// TwinCAT 3 PLC project PLC
// ProgramVersion: 3.1.4022.1
// libraries:
//   Tc2_Standard, * (Beckhoff Automation GmbH)
//   Tc2_System, * (Beckhoff Automation GmbH)
//   Tc3_Module, * (Beckhoff Automation GmbH)
// project tree:
//   DUTs/ Trapez.TcDUT, Trig.TcDUT
//   / GlobalTextList.TcGTLO, PlcTask.TcTTO, Visualization Manager.TcVMO (not stored)
//   GVLs/ IO.TcGVL, Temperatures.TcGVL
//   POUs/Fuzzy/ fbFuzzyController.TcPOU, FuzzificationTrapez.TcPOU, FuzzificationTrig.TcPOU
//   POUs/ MAIN.TcPOU, SLL.TcPOU
//   POUs/PID/ fbFlowControl.TcPOU, fbPIContoller.TcPOU, fbTempControl.TcPOU
//   POUs/utils/ fbB2U.TcPOU, fbIfElse.TcPOU, fbScale.TcPOU, fbSplit.TcPOU, fbU2B.TcPOU
// real-time tasks:
//   TASK PlcTask: cycle T#10ms, priority 20, ADS port 350
// I/O:
//   DEVICE Device 3 (EtherCAT), AmsNetId 192.168.8.100.4.1
//     Box 1 (ABB CI511) [CI511-ETHCAT (4AI 2AO 8DI 8DO)]
//     Box 2 (ABB CI512) [CI512-ETHCAT (8DC 8DI 8DO)]
// variable links:
//   PLC/PLC Instance <-> Device 3 (EtherCAT)/Box 1 (ABB CI511)
//     PlcTask Inputs/IO.AI0_Temp <-> Inputs/AI 0
//     PlcTask Inputs/IO.AI1_Pres <-> Inputs/AI 1
//     PlcTask Outputs/IO.AO0_Fan <-> Outputs/AO 0
//     PlcTask Outputs/IO.AO1_Heater <-> Outputs/AO 1
//   PLC/PLC Instance <-> Device 3 (EtherCAT)/Box 2 (ABB CI512)
//     PlcTask Inputs/IO.DI_SLL <-> Inputs/DI
//     PlcTask Outputs/IO.DO_SLL <-> Outputs/DO

CONFIGURATION PLC
    RESOURCE PLC ON TwinCAT3
        TASK PlcTask(INTERVAL := T#10ms, PRIORITY := 20);
        PROGRAM MAIN WITH PlcTask : MAIN;
    END_RESOURCE
END_CONFIGURATION

// ---- DUTs/Trapez.TcDUT
TYPE Trapez :
STRUCT
	A	:REAL;
	B	:REAL;
	C	:REAL;
	D	:REAL;
END_STRUCT
END_TYPE

// ---- DUTs/Trig.TcDUT
TYPE Trig :
STRUCT
	A	:REAL;
	B	:REAL;
	C	:REAL;
END_STRUCT
END_TYPE

// ---- GVLs/IO.TcGVL
{attribute 'qualified_only'}
VAR_GLOBAL
	AI0_Temp 	AT %I*: INT;	//Temperature
	AI1_Pres 	AT %I*:	INT;	//Pressure
	AO0_Fan 	AT %Q*: INT;	//Fan
	AO1_Heater	AT %Q*:	INT;	//Heater
	DI_SLL		AT %I*: UINT;	//Digital input
	DO_SLL		AT %Q*: UINT;	//Digital output	
END_VAR

// ---- GVLs/Temperatures.TcGVL
{attribute 'qualified_only'}
VAR_GLOBAL
	T_Ref	:REAL := 40;
	T_Act	:REAL;
END_VAR

// ---- POUs/MAIN.TcPOU
PROGRAM MAIN
VAR
	HeaterRatio			:REAL	:= 20;
	FanRatio			:REAL;
	Region				:REAL	:= 2.5; //Allowed error +- for the steady-state
	
	fbTempScale			:fbScale;
	fbFControl			:fbFuzzyController;
	fbPIControl			:fbPIContoller;
	
	Timer				:TON;
END_VAR

//Handle digital I/O
SLL(SteadyStateRegion := Region);

//HeaterRatio can be cnaged from the GUI
IO.AO1_Heater := REAL_TO_INT(27468 * HeaterRatio/100);
//Used in the GUI
FanRatio := INT_TO_REAL(IO.AO0_Fan)/INT_TO_REAL(27468)*100;


//Run the controller
//Controller can be switched between PI and Fuzzy
IF SLL.ControllerSwitch THEN
	//Longer samplingtime allows error to accumulate
	//10ms had too small changes between samples
	Timer(IN := NOT Timer.Q, PT := T#0.1S);
	IF Timer.Q THEN
		fbFControl(On := SLL.ControllerOn);
	END_IF
ELSE
	fbPIControl(On := SLL.ControllerOn);
END_IF

//Current temperature as celsius
fbTempScale(IN := IO.AI0_Temp, Scale_L := 20, Scale_H := 120);
Temperatures.T_Act := fbTempScale.OUT;

END_PROGRAM

// ---- POUs/utils/fbScale.TcPOU
FUNCTION_BLOCK fbScale
VAR_INPUT
	IN		:REAL;
	Scale_L	:REAL;
	Scale_H	:REAL;
	bType	:BOOL	:=TRUE;	//TRUE = analog val to real, FALSE = real to analog
END_VAR
VAR_OUTPUT
	OUT		:REAL;
END_VAR
VAR
	AnalogMax :REAL := 27648;
END_VAR

IF bType THEN
	OUT := IN / AnalogMax * (Scale_H - Scale_L) + Scale_L;
ELSE
	OUT := (AnalogMax * (IN - Scale_L)) / (Scale_H - Scale_L);
END_IF

END_FUNCTION_BLOCK

// ---- POUs/Fuzzy/fbFuzzyController.TcPOU
FUNCTION_BLOCK fbFuzzyController
VAR_INPUT
	On					:BOOL;
END_VAR
VAR_OUTPUT
END_VAR
VAR
	HOT, COLD						:Trapez;
	WARM, COOL						:Trig;
	
	DECREASING, INCREASING			:Trapez;
	SLOWDOWN, SPEEDUP				:Trig;
	
	Temperature						:REAL;
	Temp_prev						:REAL := 0;
	Error							:REAL := 0;
	
	//Degree of membership
	Hot_h, Warm_h, Cool_h, Cold_h	:REAL;
	Decreasing_h, Increasing_h		:REAL;
	
	Rule, Rule1, Rule2, Rule3, Rule4, Rule5, Rule6 :REAL;
	
	u	:REAL;
	Fan_R	:REAL;
	Scale	:REAL := 0.1;
END_VAR

//If controller is switched off, turn the fan off and reset the controllers
IF NOT On THEN
	IO.AO0_Fan := 0;
	RETURN;
END_IF

//Temperature
HOT.A := -100; HOT.B := -100; HOT.C := -5; HOT.D := -0.5;
WARM.A := -5; WARM.B := -2.5; WARM.C := 0;
COOL.A := 0; COOL.B := 2.5; COOL.C := 5;
COLD.A := 0.5; COLD.B := 5; COLD.C := 100; COLD.D := 100;

//Error
DECREASING.A := -0.1; DECREASING.B := -0.03; DECREASING.C := -0.0006; DECREASING.D := 0;
INCREASING.A := 0; INCREASING.B := 0.0006; INCREASING.C := 0.03; INCREASING.D := 0.1;

//Control signal
SLOWDOWN.A := 1; SLOWDOWN.B := -1; SLOWDOWN.C := -1;
SPEEDUP.A := -1; SPEEDUP.B := 1; SPEEDUP.C := 1;

//Controller inputs
Temperature := Temperatures.T_Ref - Temperatures.T_Act;
Error := Temp_prev - Temperature;
Temp_prev := Temperature;

//Fuzzification
Hot_h := FuzzificationTrapez(Temperature, HOT);
Cold_h := FuzzificationTrapez(Temperature, COLD);
Warm_h := FuzzificationTrig(Temperature, WARM);
Cool_h := FuzzificationTrig(Temperature, Cool);
Decreasing_h := FuzzificationTrapez(Error, DECREASING);
Increasing_h := FuzzificationTrapez(Error, INCREASING);

//Rules
//IF Temperature IS Hot
IF Hot_h > 0 THEN
	Rule1 := Hot_h;
END_IF
//IF Temperature IS Warm AND Error IS Increasing
IF Warm_h > 0 AND Increasing_h > 0 THEN
	Rule2 := MIN(Warm_h,Increasing_h);
END_IF
//IF Temperature IS Warm AND Error IS Decreasing
IF Warm_h > 0 AND Decreasing_h > 0 THEN
	Rule3 := MIN(Warm_h,Decreasing_h);
END_IF
//IF Temperature IS Cool AND Error IS Increasing
IF Cool_h > 0 AND Increasing_h > 0 THEN
	Rule4 := MIN(Cool_h,Increasing_h);
END_IF
//IF Temperature IS Cool AND Error IS Decreasing
IF Cool_h > 0 AND Decreasing_h > 0 THEN
	Rule5 := MIN(Cool_h,Decreasing_h);
END_IF
//IF Temperature IS Cold
IF Cold_h > 0 THEN
	Rule6 := Cold_h;
END_IF

//Rule with the max value is the most significant
Rule := MAX(Rule1,Rule2,Rule3,Rule4,Rule5,Rule6);

//Defuzzification using Mean of Max.
//Boundaries with alpha-cut at max rule's degree
IF Rule = Rule1 OR Rule = Rule2 OR Rule = Rule4 THEN
	u := ((SPEEDUP.B-SPEEDUP.A)*Rule+SPEEDUP.A + (-(SPEEDUP.C-SPEEDUP.B)*Rule+SPEEDUP.C))/2;
ELSIF Rule = Rule3 OR Rule = Rule5 OR Rule = Rule6 THEN
	u := ((SLOWDOWN.B-SLOWDOWN.A)*Rule+SLOWDOWN.A + (-(SLOWDOWN.C-SLOWDOWN.B)*Rule+SLOWDOWN.C))/2;
END_IF
//Resetting values to zero for the next execution
Rule1 := Rule2 := Rule3 := Rule4 := Rule5 := Rule6 := 0;

//Calculating the new fan usage 0-100
Fan_R := Fan_R + u * Scale;
IF Fan_R > 100 THEN
	Fan_R := 100;
ELSIF FAN_R < 0 THEN
	Fan_R := 0;
END_IF

IO.AO0_Fan := REAL_TO_INT(27648*Fan_R/100);

END_FUNCTION_BLOCK

// ---- POUs/Fuzzy/FuzzificationTrapez.TcPOU
FUNCTION FuzzificationTrapez : REAL
VAR_INPUT
	x		:REAL;
	trapez	:Trapez;
END_VAR
VAR
END_VAR

IF x <= trapez.A THEN
	FuzzificationTrapez := 0;
ELSIF trapez.A < x AND x <= trapez.B THEN
	FuzzificationTrapez := (x-trapez.A)/(trapez.B-trapez.A);
ELSIF trapez.B <= x AND x <= trapez.C THEN
	FuzzificationTrapez := 1;
ELSIF trapez.C < x AND x <= trapez.D THEN
	FuzzificationTrapez := (trapez.D-x)/(trapez.D-trapez.C);
ELSIF trapez.D < x THEN
	FuzzificationTrapez := 0; 
END_IF

END_FUNCTION

// ---- POUs/Fuzzy/FuzzificationTrig.TcPOU
FUNCTION FuzzificationTrig : REAL
VAR_INPUT
	x		:REAL;
	trig	:Trig;
END_VAR
VAR
END_VAR

IF x <= trig.A THEN
	FuzzificationTrig := 0;
ELSIF trig.A < x AND x <= trig.B THEN
	FuzzificationTrig := (x-trig.A)/(trig.B-trig.A);
ELSIF trig.B < x AND x <= trig.C THEN
	FuzzificationTrig := (trig.C-x)/(trig.C-trig.B);
ELSIF trig.C < x THEN
	FuzzificationTrig := 0; 
END_IF

END_FUNCTION

// ---- POUs/PID/fbPIContoller.TcPOU
FUNCTION_BLOCK fbPIContoller
VAR_INPUT
	On					:BOOL;
END_VAR
VAR
	//PID-variables
	P_Temperature		:REAL	:= 10.0;
	P_Flow				:REAL	:= 2.0;
	Ki_Temperature		:REAL 	:= 0.005;
	Ki_Flow				:REAL 	:= 0.001;
	I_CapTemperature	:INT	:= 80;
	I_CapFlow			:INT	:= 80;

	//FBs

	fbFlowScale			:fbScale;
	fbFlowP2AScale		:fbScale;
	
	fbFlowController	:fbFlowControl;
	fbTempController	:fbTempControl;
END_VAR

//If controller is switched off, turn the fan off and reset the controllers
IF NOT On THEN
	IO.AO0_Fan := 0;
	RETURN;
END_IF

//Current flowrate
fbFlowScale(IN := IO.AI1_Pres, Scale_L := 0, Scale_H := 100);

fbTempController(
	Act := Temperatures.T_Act,
	Ref := Temperatures.T_Ref,
	Kp := P_Temperature,
	Ki := Ki_Temperature,
	I_Cap := I_CapTemperature);

fbFlowController(
	Act := fbFlowScale.OUT,
	Ref := fbTempController.OUT,
	Kp := P_Flow,
	Ki := Ki_Flow,
	I_Cap := I_CapFlow);

//Percentage to analog value (0-100% -> 0-27468)
fbFlowP2AScale(IN := fbFlowController.OUT, Scale_L := 0, Scale_H := 100, bType := FALSE);
IO.AO0_Fan := REAL_TO_INT(fbFlowP2AScale.OUT);

END_FUNCTION_BLOCK

// ---- POUs/PID/fbFlowControl.TcPOU
FUNCTION_BLOCK fbFlowControl
VAR_INPUT
	Act			:REAL; //0 - 27846
	Ref			:REAL; //0 - 27846
	Kp			:REAL;
	Ki			:REAL;
	I_Cap		:INT; //Maximum value of the Integral portion
END_VAR
VAR_OUTPUT
	OUT			:INT;
END_VAR
VAR
	Error 		:REAL;
	P_Out		:REAL;
	I_Out		:REAL;
	PI_Out		:REAL;
END_VAR

Error :=  Ref - Act;
P_Out := Kp * Error;
I_Out := Ki * Error + I_Out;

IF I_Out > I_Cap THEN
	I_Out := I_Cap;
END_IF

PI_Out := P_Out + I_Out;

IF PI_Out > 100 THEN
	OUT := 100;
ELSIF PI_Out < 5 THEN
	//Small amount of flow to make temperature rise more evenly
	//inside the tube
	OUT := 5;
ELSE
	//IO requires INT => conversion from real to int
	OUT := REAL_TO_INT(PI_Out);
END_IF

END_FUNCTION_BLOCK

// ---- POUs/PID/fbTempControl.TcPOU
FUNCTION_BLOCK fbTempControl
VAR_INPUT
	Act			:REAL; //Celsius
	Ref			:REAL; //Celsius
	Kp			:REAL;
	Ki			:REAL;
	I_Cap		:INT; //Maximum value of the Integral portion
END_VAR
VAR_OUTPUT
	OUT			:REAL;
END_VAR
VAR
	Error 		:REAL;
	P_Out		:REAL;
	I_Out		:REAL;
	PI_Out		:REAL;
	AnalogMax	:INT	:= 27846;
END_VAR

Error :=  Act - Ref;
P_Out := Kp * Error;
I_Out := Ki * Error + I_Out;

IF I_Out > I_Cap THEN
	I_Out := I_Cap;
ELSIF I_Out < 0 THEN
	I_Out := 0;
END_IF

PI_Out := P_Out + I_Out;

//100 is the maximum sensor value
IF PI_Out > 100 THEN
	OUT := 100;
ELSIF PI_Out < 0 THEN
	OUT := 0;
ELSE
	OUT := PI_Out;
END_IF

END_FUNCTION_BLOCK

// ---- POUs/SLL.TcPOU
PROGRAM SLL
VAR_INPUT
	SteadyStateRegion	:REAL;
END_VAR
VAR_OUTPUT
	ControllerOn		:BOOL;
	ControllerSwitch	:BOOL;
END_VAR
VAR
	u2b			:fbU2B;
	b2u			:fbB2U;
	split1		:fbSplit;
	split2		:fbSplit;
	r_trigu		:R_TRIG;
	r_trigd		:R_TRIG;
	IfElse1		:fbIfElse;
	IfElse2		:fbIfElse;
END_VAR
VAR // added by the converter: edge detectors and wires of the graphical bodies
    _w1, _w2 : BOOL;
    _w3 : ANY;
END_VAR


// PAGE -1
// Calculating weather the system is in steadystate or not
_w1 := ABS(Temperatures.T_Act - Temperatures.T_Ref) < SteadyStateRegion;
// Fan is on/off
_w2 := NOT (IO.AO0_Fan = 0);
// Switch between Fuzzy and PI
ControllerSwitch := u2b.B5;
u2b(IN := IO.DI_SLL); // fbU2B
// If the switch is on, set red LED off
// and start the controller
split1(IN := BOOL_TO_REAL(u2b.B4)); // fbSplit
// Switch LEDs on/off
b2u(B1 := NOT REAL_TO_BOOL(split1.OUT1), B2 := _w1, B3 := _w2); // fbB2U
IO.DO_SLL := b2u.OUT;
ControllerOn := REAL_TO_BOOL(split1.OUT2);
// Add 1 to the reference temperature, if the button is pressed
r_trigu(CLK := u2b.B1); // R_TRIG
split2(IN := Temperatures.T_Ref); // fbSplit
// If button is pressed and the
// trigger sends true, the ref + 1
// value is set as output.
// Otherwise it stays as ref
IfElse1(BVal := r_trigu.Q, IFVal := 1 + split2.OUT1, ELSEVal := Temperatures.T_Ref); // fbIfElse
_w3 := split2.OUT2 - 1;
// If button is pressed and the trigger sends true,
// the ref -1 is set as output.
// Otherwise the value from IfElse1 is set as output.
// Substract 1 from the reference temperature, if the button is pressed
r_trigd(CLK := u2b.B2); // R_TRIG
IfElse2(BVal := r_trigd.Q, IFVal := _w3, ELSEVal := IfElse1.OUT); // fbIfElse
Temperatures.T_Ref := IfElse2.OUT;

END_PROGRAM

// ---- POUs/utils/fbU2B.TcPOU
FUNCTION_BLOCK fbU2B
VAR_INPUT
	IN		:UINT;
END_VAR
VAR_OUTPUT
	B1		:BOOL;
	B2		:BOOL;
	B3		:BOOL;
	B4		:BOOL;
	B5		:BOOL;
END_VAR
VAR
	Index	:INT;
	D_val	:UINT;
	Rem		:UINT := 0;
END_VAR

//Turning the digial input into five booleans
//First 8 bits are always zeros so the first needed boolean value is at index 8 (zero based)
D_val := IN;
FOR Index := 0 TO 12 DO
	Rem := D_val MOD 2;
	D_val := (D_val-Rem) / 2;
	IF Index = 8 THEN
		B1 := UINT_TO_BOOL(Rem);
	ELSIF Index = 9 THEN
		B2 := UINT_TO_BOOL(Rem);
	ELSIF Index = 10 THEN
		B3 := UINT_TO_BOOL(Rem);
	ELSIF Index = 11 THEN
		B4 := UINT_TO_BOOL(Rem);
	ELSIF Index = 12 THEN
		B5 := UINT_TO_BOOL(Rem);
	END_IF
END_FOR

END_FUNCTION_BLOCK

// ---- POUs/utils/fbB2U.TcPOU
FUNCTION_BLOCK fbB2U
VAR_INPUT
	B1		:BOOL;
	B2		:BOOL;
	B3		:BOOL;
	B4		:BOOL;
END_VAR
VAR_OUTPUT
	OUT		:UINT;
END_VAR
VAR
	B_Arr	:ARRAY [0 .. 3] OF BOOL;
	D_val	:UINT;
	Index	:INT;
	Pow		:INT;
END_VAR

//Turning 12 bits into an integer
//First 8 bits are zeros, so the Pow starts at 8
Pow := 8;
D_Val := 0;
B_Arr[0] := B1;
B_Arr[1] := B2;
B_Arr[2] := B3;
B_Arr[3] := B4;
FOR Index := 0 TO 3 DO
	D_Val := LREAL_TO_UINT(D_Val + BOOL_TO_INT(B_Arr[Index])*EXPT(2,Pow));
	Pow := Pow + 1;
END_FOR
OUT := D_Val;

END_FUNCTION_BLOCK

// ---- POUs/utils/fbSplit.TcPOU
FUNCTION_BLOCK fbSplit
VAR_INPUT
	IN		:REAL;
END_VAR
VAR_OUTPUT
	OUT1	:REAL;
	OUT2	:REAL;
END_VAR
VAR
END_VAR

//Split one input into two outputs
OUT1 := IN;
OUT2 := IN;

END_FUNCTION_BLOCK

// ---- POUs/utils/fbIfElse.TcPOU
FUNCTION_BLOCK fbIfElse
VAR_INPUT
	BVal		:BOOL;
	IFVal		:REAL;
	ELSEVal		:REAL;
END_VAR
VAR_OUTPUT
	OUT			:REAL;
END_VAR
VAR
END_VAR

IF BVal THEN
	OUT := IFVal;
ELSE
	OUT := ELSEVal;
END_IF

END_FUNCTION_BLOCK
